(* Logix 5000 project; controller NSH_PLC2 vendor 1 type 14 code 167 rev 32.14; software revision 32.03; part 6 of 6 *)
(* tags used below, declared in another part *)
   AFI : BOOL;   // Always False
   AOI_PLC1_To_MCC3_10A : MotorToE300;
   AOI_PLC1_To_MCC3_10D : MotorToE300;
   AOI_PLC1_To_MCC3_10G : MotorToE300;
   AOI_PLC1_To_MCC3_10J : MotorToE300;
   AOI_PLC1_To_MCC3_11A : MotorToE300;
   AOI_PLC1_To_MCC3_11D : MotorToE300;
   AOI_PLC1_To_MCC3_11G : MotorToE300;
   AOI_PLC1_To_MCC3_11J : MotorToE300;
   AOI_PLC1_To_MCC3_12A : MotorToE300;
   AOI_PLC1_To_MCC3_12C : MotorToE300;
   AOI_PLC1_To_MCC3_12E : MotorToE300;
   AOI_PLC1_To_MCC3_12G : MotorToE300;
   AOI_PLC1_To_MCC3_12J : MotorToE300;
   AOI_PLC1_To_MCC3_12L : MotorToE300;
   AOI_PLC1_To_MCC3_13A : MotorToE300;
   AOI_PLC1_To_MCC3_13C : MotorToE300;
   AOI_PLC1_To_MCC3_13E : MotorToE300;
   AOI_PLC1_To_MCC3_13G : MotorToE300;
   AOI_PLC1_To_MCC3_13J : MotorToE300;
   AOI_PLC1_To_MCC3_13L : MotorToE300;
   AOI_PLC1_To_MCC3_14A : MotorToE300;
   AOI_PLC1_To_MCC3_14C : MotorToE300;
   AOI_PLC1_To_MCC3_14E : MotorToE300;
   AOI_PLC1_To_MCC3_14G : MotorToE300;
   AOI_PLC1_To_MCC3_14J : MotorToE300;
   AOI_PLC1_To_MCC3_14L : MotorToE300;
   AOI_PLC1_To_MCC3_15A : MotorToE300;
   AOI_PLC1_To_MCC3_15C : MotorToE300;
   AOI_PLC1_To_MCC3_15E : MotorToE300;
   AOI_PLC1_To_MCC3_15G : MotorToE300;
   AOI_PLC1_To_MCC3_15J : MotorToE300;
   AOI_PLC1_To_MCC3_16A : MotorToE300;
   AOI_PLC1_To_MCC3_16C : MotorToE300;
   AOI_PLC1_To_MCC3_16E : MotorToE300;
   AOI_PLC1_To_MCC3_16G : MotorToE300;
   AOI_PLC1_To_MCC3_16J : MotorToE300;
   AOI_PLC1_To_MCC3_16L : MotorToE300;
   AOI_PLC1_To_MCC3_17A : MotorToE300;
   AOI_PLC1_To_MCC3_17C : MotorToE300;
   AOI_PLC1_To_MCC3_17E : MotorToE300;
   AOI_PLC1_To_MCC3_17G : MotorToE300;
   AOI_PLC1_To_MCC3_17J : MotorToE300;
   AOI_PLC1_To_MCC3_17L : MotorToE300;
   AOI_PLC1_To_MCC3_18A : MotorToE300;
   AOI_PLC1_To_MCC3_18C : MotorToE300;
   AOI_PLC1_To_MCC3_18E : MotorToE300;
   AOI_PLC1_To_MCC3_18G : MotorToE300;
   AOI_PLC1_To_MCC3_18J : MotorToE300;
   AOI_PLC1_To_MCC3_18L : MotorToE300;
   AOI_PLC1_To_MCC3_19A : MotorToE300;
   AOI_PLC1_To_MCC3_19C : MotorToE300;
   AOI_PLC1_To_MCC3_19E : MotorToE300;
   AOI_PLC1_To_MCC3_19G : MotorToE300;
   AOI_PLC1_To_MCC3_19J : MotorToE300;
   AOI_PLC1_To_MCC3_20A : MotorToE300;
   AOI_PLC1_To_MCC3_20C : MotorToE300;
   AOI_PLC1_To_MCC3_20E : MotorToE300;
   AOI_PLC1_To_MCC3_20G : MotorToE300;
   AOI_PLC1_To_MCC3_20J : MotorToE300;
   AOI_PLC1_To_MCC3_21A : MotorToE300;
   AOI_PLC1_To_MCC3_21C : MotorToE300;
   AOI_PLC1_To_MCC3_21E : MotorToE300;
   AOI_PLC1_To_MCC3_21G : MotorToE300;
   AOI_PLC1_To_MCC3_21J : MotorToE300;
   AOI_PLC1_To_MCC3_21L : MotorToE300;
   AOI_PLC1_To_MCC3_22C : MotorToE300;
   AOI_PLC1_To_MCC3_22E : MotorToE300;
   AOI_PLC1_To_MCC3_7A : MotorToE300;
   AOI_PLC1_To_MCC3_7C : MotorToE300;
   AOI_PLC1_To_MCC3_7E : MotorToE300;
   AOI_PLC1_To_MCC3_7G : MotorToPF525;
   AOI_PLC1_To_MCC3_7K : MotorToPF525;
   AOI_PLC1_To_MCC3_8A : MotorToE300;
   AOI_PLC1_To_MCC3_8D : MotorToPF525;
   AOI_PLC1_To_MCC3_8H : MotorToE300;
   AOI_PLC1_To_MCC3_8K : MotorToPF525;
   AOI_PLC1_To_MCC3_9A : MotorToE300;
   AOI_PLC1_To_MCC3_9C : MotorToE300;
   AOI_PLC1_To_MCC3_9E : MotorToE300;
   AOI_PLC1_To_MCC3_9G : MotorToE300;
   AOI_PLC1_To_MCC3_9J : MotorToE300;
   AOI_PLC1_To_MCC3_9L : MotorToE300;
   AOI_PLC1_To_MCC4_1E : MotorToPF525;
   AOI_PLC1_To_MCC4_2A : MotorToE300;
   AOI_PLC1_To_MCC4_2C : MotorToE300;
   AOI_PLC1_To_MCC4_2E : MotorToE300;
   AOI_PLC1_To_MCC4_2G : MotorToPF525;
   AOI_PLC1_To_MCC4_2K : MotorToPF525;
   AOI_PLC1_To_MCC4_3A : MotorToE300;
   AOI_PLC1_To_MCC4_3C : MotorToE300;
   AOI_PLC1_To_MCC4_3E : MotorToE300;
   AOI_PLC1_To_MCC4_3G : MotorToE300;
   AOI_PLC1_To_MCC4_3J : MotorToE300;
   AOI_PLC1_To_MCC4_3L : MotorToE300;
   AOI_PLC1_To_MCC4_4A : MotorToE300;
   AOI_PLC1_To_MCC4_4C : MotorToE300;
   AOI_PLC1_To_MCC4_4E : MotorToE300;
   AOI_PLC1_To_MCC4_4G : MotorToE300;
   AOI_PLC1_To_MCC4_4J : MotorToE300;
   AOI_PLC1_To_MCC4_4L : MotorToE300;
   AOI_PLC1_To_MCC4_5A : MotorToE300;
   AOI_PLC1_To_MCC4_5C : MotorToE300;
   MotorsControlTag : MotorsControlUDT;   // Only Instance of UDT
   OKToRunMotors : BOOL;   // Messages from PLC1 Ok, OK to run
(* MainProgram, continued *)

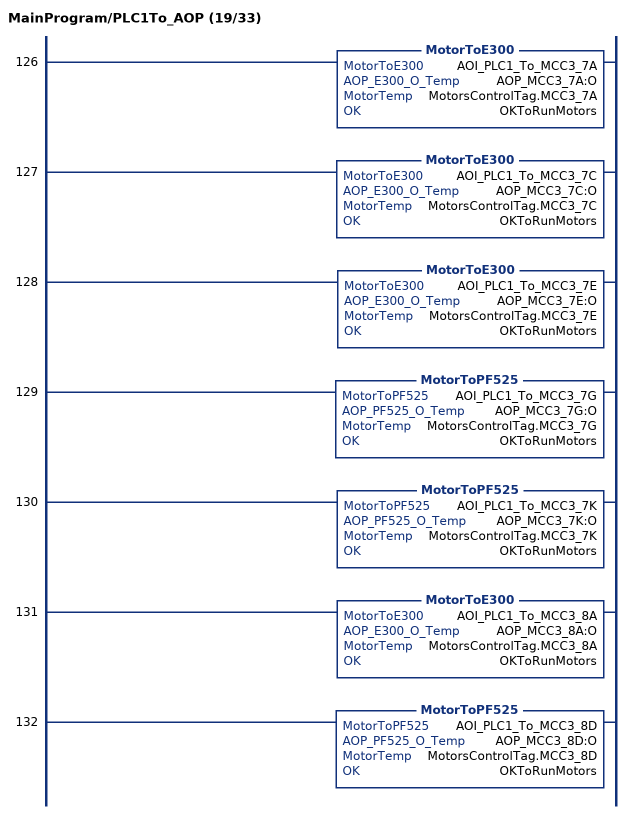
   [picture p103: MainProgram/PLC1To_AOP rungs 126-132]
   126: MotorToE300(AOI_PLC1_To_MCC3_7A,AOP_MCC3_7A:O,MotorsControlTag.MCC3_7A,OKToRunMotors);
   127: MotorToE300(AOI_PLC1_To_MCC3_7C,AOP_MCC3_7C:O,MotorsControlTag.MCC3_7C,OKToRunMotors);
   128: MotorToE300(AOI_PLC1_To_MCC3_7E,AOP_MCC3_7E:O,MotorsControlTag.MCC3_7E,OKToRunMotors);
   129: MotorToPF525(AOI_PLC1_To_MCC3_7G,AOP_MCC3_7G:O,MotorsControlTag.MCC3_7G,OKToRunMotors);
   130: MotorToPF525(AOI_PLC1_To_MCC3_7K,AOP_MCC3_7K:O,MotorsControlTag.MCC3_7K,OKToRunMotors);
   131: MotorToE300(AOI_PLC1_To_MCC3_8A,AOP_MCC3_8A:O,MotorsControlTag.MCC3_8A,OKToRunMotors);
   132: MotorToPF525(AOI_PLC1_To_MCC3_8D,AOP_MCC3_8D:O,MotorsControlTag.MCC3_8D,OKToRunMotors);
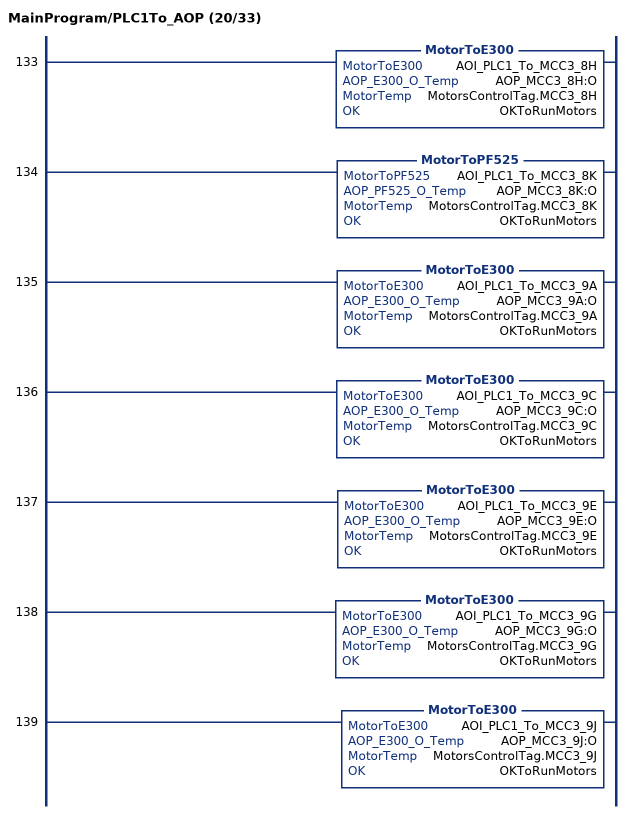
   133: MotorToE300(AOI_PLC1_To_MCC3_8H,AOP_MCC3_8H:O,MotorsControlTag.MCC3_8H,OKToRunMotors);
   134: MotorToPF525(AOI_PLC1_To_MCC3_8K,AOP_MCC3_8K:O,MotorsControlTag.MCC3_8K,OKToRunMotors);
   135: MotorToE300(AOI_PLC1_To_MCC3_9A,AOP_MCC3_9A:O,MotorsControlTag.MCC3_9A,OKToRunMotors);
   136: MotorToE300(AOI_PLC1_To_MCC3_9C,AOP_MCC3_9C:O,MotorsControlTag.MCC3_9C,OKToRunMotors);
   137: MotorToE300(AOI_PLC1_To_MCC3_9E,AOP_MCC3_9E:O,MotorsControlTag.MCC3_9E,OKToRunMotors);
   138: MotorToE300(AOI_PLC1_To_MCC3_9G,AOP_MCC3_9G:O,MotorsControlTag.MCC3_9G,OKToRunMotors);
   139: MotorToE300(AOI_PLC1_To_MCC3_9J,AOP_MCC3_9J:O,MotorsControlTag.MCC3_9J,OKToRunMotors);
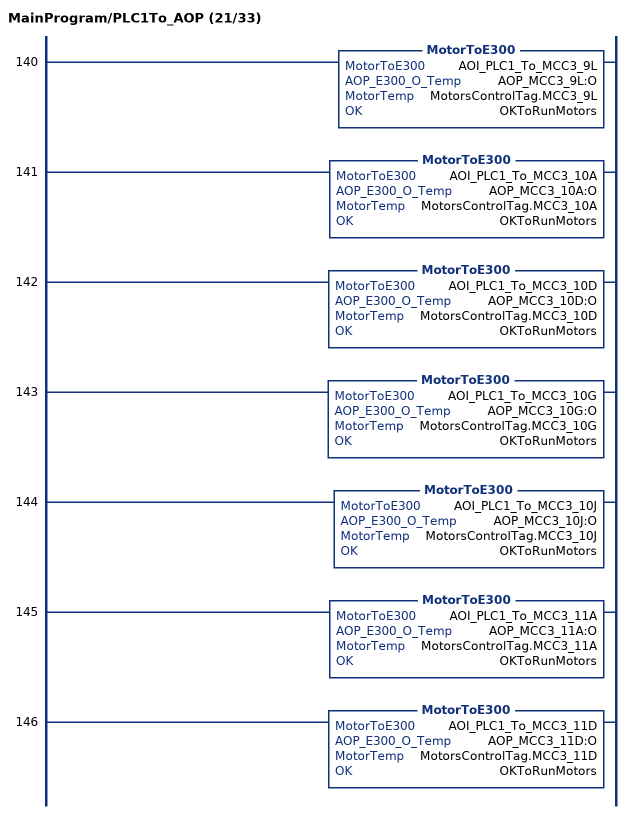
   140: MotorToE300(AOI_PLC1_To_MCC3_9L,AOP_MCC3_9L:O,MotorsControlTag.MCC3_9L,OKToRunMotors);
   141: MotorToE300(AOI_PLC1_To_MCC3_10A,AOP_MCC3_10A:O,MotorsControlTag.MCC3_10A,OKToRunMotors);
   142: MotorToE300(AOI_PLC1_To_MCC3_10D,AOP_MCC3_10D:O,MotorsControlTag.MCC3_10D,OKToRunMotors);
   143: MotorToE300(AOI_PLC1_To_MCC3_10G,AOP_MCC3_10G:O,MotorsControlTag.MCC3_10G,OKToRunMotors);
   144: MotorToE300(AOI_PLC1_To_MCC3_10J,AOP_MCC3_10J:O,MotorsControlTag.MCC3_10J,OKToRunMotors);
   145: MotorToE300(AOI_PLC1_To_MCC3_11A,AOP_MCC3_11A:O,MotorsControlTag.MCC3_11A,OKToRunMotors);
   146: MotorToE300(AOI_PLC1_To_MCC3_11D,AOP_MCC3_11D:O,MotorsControlTag.MCC3_11D,OKToRunMotors);
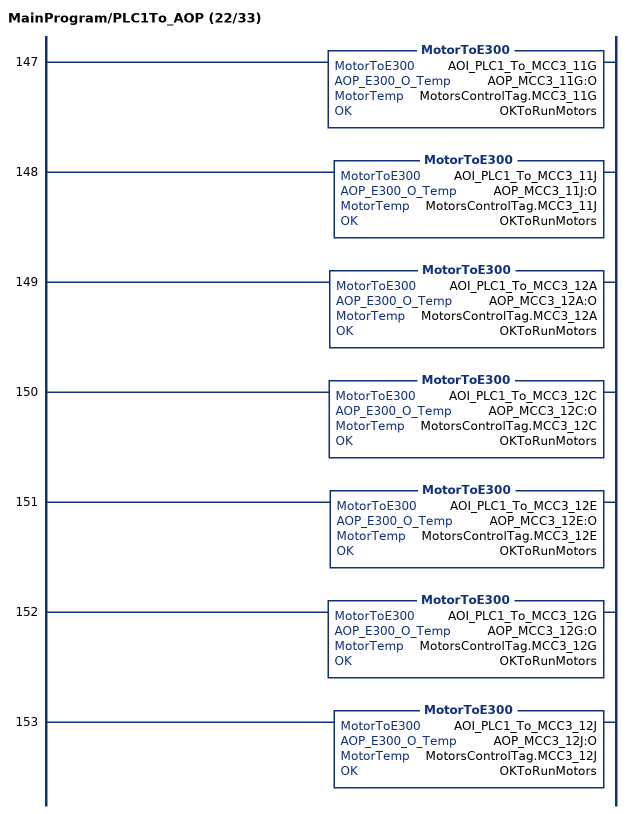
   147: MotorToE300(AOI_PLC1_To_MCC3_11G,AOP_MCC3_11G:O,MotorsControlTag.MCC3_11G,OKToRunMotors);
   148: MotorToE300(AOI_PLC1_To_MCC3_11J,AOP_MCC3_11J:O,MotorsControlTag.MCC3_11J,OKToRunMotors);
   149: MotorToE300(AOI_PLC1_To_MCC3_12A,AOP_MCC3_12A:O,MotorsControlTag.MCC3_12A,OKToRunMotors);
   150: MotorToE300(AOI_PLC1_To_MCC3_12C,AOP_MCC3_12C:O,MotorsControlTag.MCC3_12C,OKToRunMotors);
   151: MotorToE300(AOI_PLC1_To_MCC3_12E,AOP_MCC3_12E:O,MotorsControlTag.MCC3_12E,OKToRunMotors);
   152: MotorToE300(AOI_PLC1_To_MCC3_12G,AOP_MCC3_12G:O,MotorsControlTag.MCC3_12G,OKToRunMotors);
   153: MotorToE300(AOI_PLC1_To_MCC3_12J,AOP_MCC3_12J:O,MotorsControlTag.MCC3_12J,OKToRunMotors);
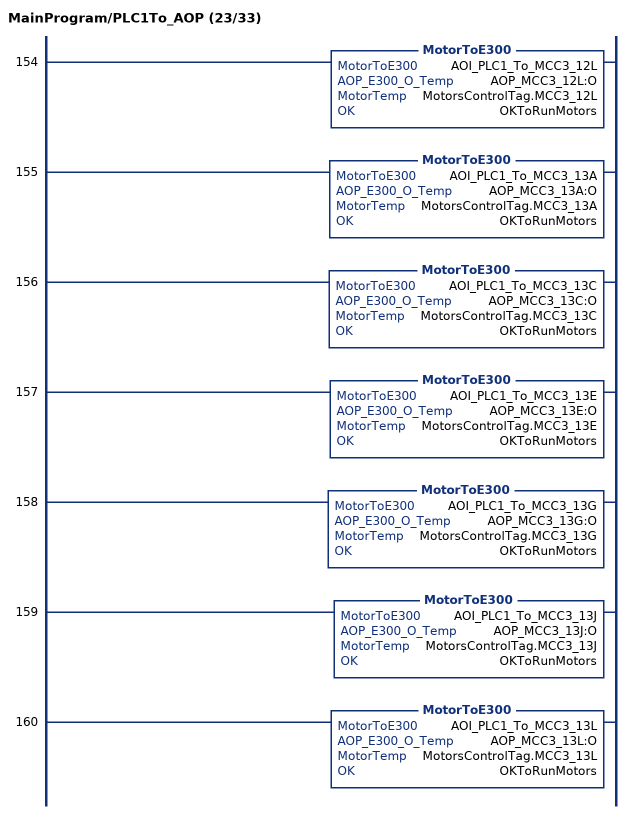
   154: MotorToE300(AOI_PLC1_To_MCC3_12L,AOP_MCC3_12L:O,MotorsControlTag.MCC3_12L,OKToRunMotors);
   155: MotorToE300(AOI_PLC1_To_MCC3_13A,AOP_MCC3_13A:O,MotorsControlTag.MCC3_13A,OKToRunMotors);
   156: MotorToE300(AOI_PLC1_To_MCC3_13C,AOP_MCC3_13C:O,MotorsControlTag.MCC3_13C,OKToRunMotors);
   157: MotorToE300(AOI_PLC1_To_MCC3_13E,AOP_MCC3_13E:O,MotorsControlTag.MCC3_13E,OKToRunMotors);
   158: MotorToE300(AOI_PLC1_To_MCC3_13G,AOP_MCC3_13G:O,MotorsControlTag.MCC3_13G,OKToRunMotors);
   159: MotorToE300(AOI_PLC1_To_MCC3_13J,AOP_MCC3_13J:O,MotorsControlTag.MCC3_13J,OKToRunMotors);
   160: MotorToE300(AOI_PLC1_To_MCC3_13L,AOP_MCC3_13L:O,MotorsControlTag.MCC3_13L,OKToRunMotors);
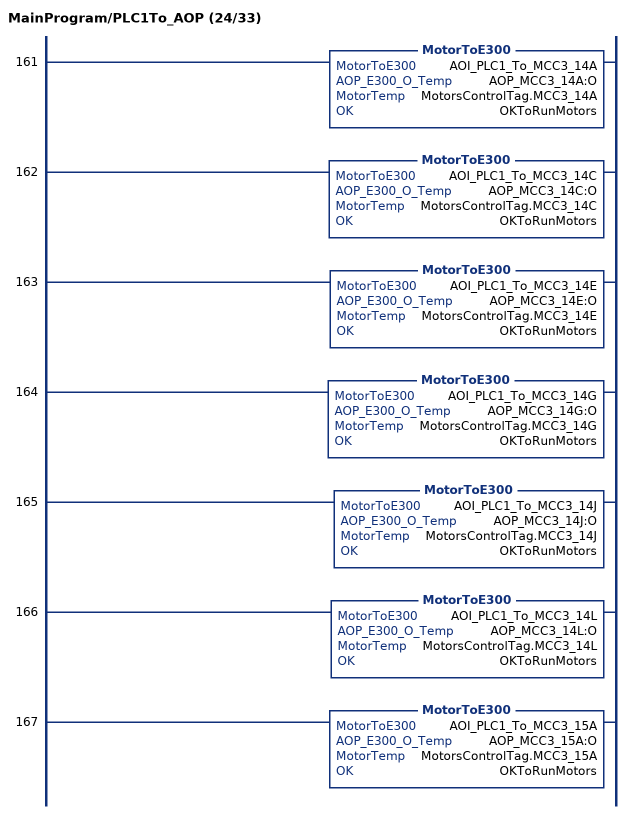
   161: MotorToE300(AOI_PLC1_To_MCC3_14A,AOP_MCC3_14A:O,MotorsControlTag.MCC3_14A,OKToRunMotors);
   162: MotorToE300(AOI_PLC1_To_MCC3_14C,AOP_MCC3_14C:O,MotorsControlTag.MCC3_14C,OKToRunMotors);
   163: MotorToE300(AOI_PLC1_To_MCC3_14E,AOP_MCC3_14E:O,MotorsControlTag.MCC3_14E,OKToRunMotors);
   164: MotorToE300(AOI_PLC1_To_MCC3_14G,AOP_MCC3_14G:O,MotorsControlTag.MCC3_14G,OKToRunMotors);
   165: MotorToE300(AOI_PLC1_To_MCC3_14J,AOP_MCC3_14J:O,MotorsControlTag.MCC3_14J,OKToRunMotors);
   166: MotorToE300(AOI_PLC1_To_MCC3_14L,AOP_MCC3_14L:O,MotorsControlTag.MCC3_14L,OKToRunMotors);
   167: MotorToE300(AOI_PLC1_To_MCC3_15A,AOP_MCC3_15A:O,MotorsControlTag.MCC3_15A,OKToRunMotors);
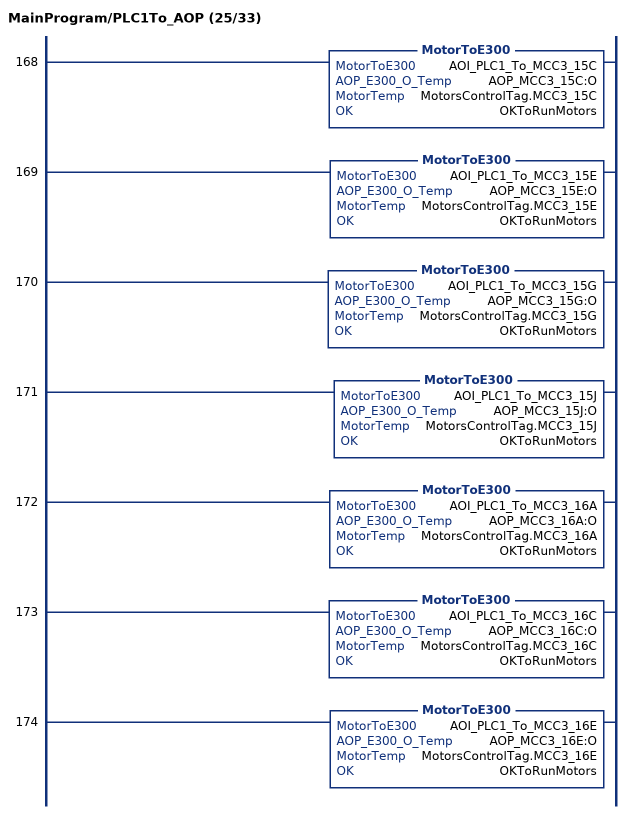
   168: MotorToE300(AOI_PLC1_To_MCC3_15C,AOP_MCC3_15C:O,MotorsControlTag.MCC3_15C,OKToRunMotors);
   169: MotorToE300(AOI_PLC1_To_MCC3_15E,AOP_MCC3_15E:O,MotorsControlTag.MCC3_15E,OKToRunMotors);
   170: MotorToE300(AOI_PLC1_To_MCC3_15G,AOP_MCC3_15G:O,MotorsControlTag.MCC3_15G,OKToRunMotors);
   171: MotorToE300(AOI_PLC1_To_MCC3_15J,AOP_MCC3_15J:O,MotorsControlTag.MCC3_15J,OKToRunMotors);
   172: MotorToE300(AOI_PLC1_To_MCC3_16A,AOP_MCC3_16A:O,MotorsControlTag.MCC3_16A,OKToRunMotors);
   173: MotorToE300(AOI_PLC1_To_MCC3_16C,AOP_MCC3_16C:O,MotorsControlTag.MCC3_16C,OKToRunMotors);
   174: MotorToE300(AOI_PLC1_To_MCC3_16E,AOP_MCC3_16E:O,MotorsControlTag.MCC3_16E,OKToRunMotors);
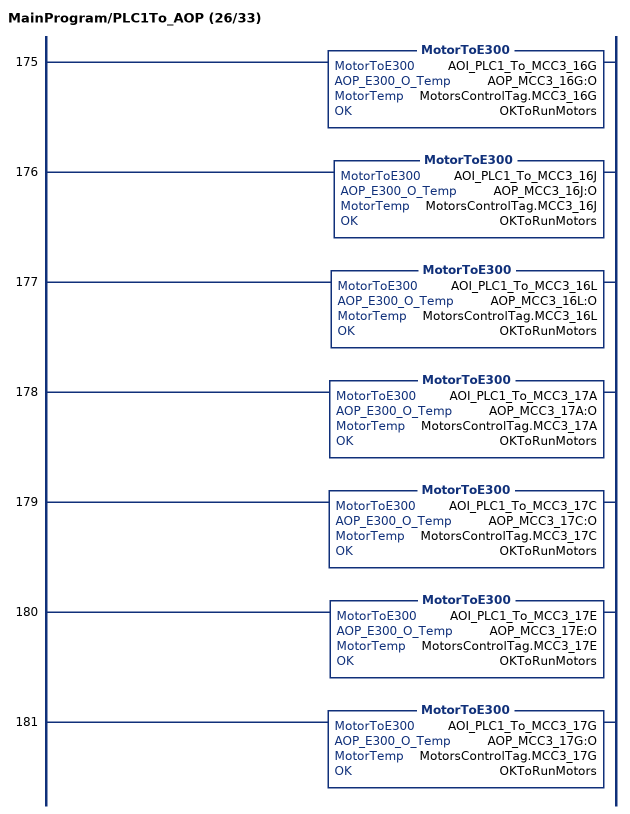
   175: MotorToE300(AOI_PLC1_To_MCC3_16G,AOP_MCC3_16G:O,MotorsControlTag.MCC3_16G,OKToRunMotors);
   176: MotorToE300(AOI_PLC1_To_MCC3_16J,AOP_MCC3_16J:O,MotorsControlTag.MCC3_16J,OKToRunMotors);
   177: MotorToE300(AOI_PLC1_To_MCC3_16L,AOP_MCC3_16L:O,MotorsControlTag.MCC3_16L,OKToRunMotors);
   178: MotorToE300(AOI_PLC1_To_MCC3_17A,AOP_MCC3_17A:O,MotorsControlTag.MCC3_17A,OKToRunMotors);
   179: MotorToE300(AOI_PLC1_To_MCC3_17C,AOP_MCC3_17C:O,MotorsControlTag.MCC3_17C,OKToRunMotors);
   180: MotorToE300(AOI_PLC1_To_MCC3_17E,AOP_MCC3_17E:O,MotorsControlTag.MCC3_17E,OKToRunMotors);
   181: MotorToE300(AOI_PLC1_To_MCC3_17G,AOP_MCC3_17G:O,MotorsControlTag.MCC3_17G,OKToRunMotors);
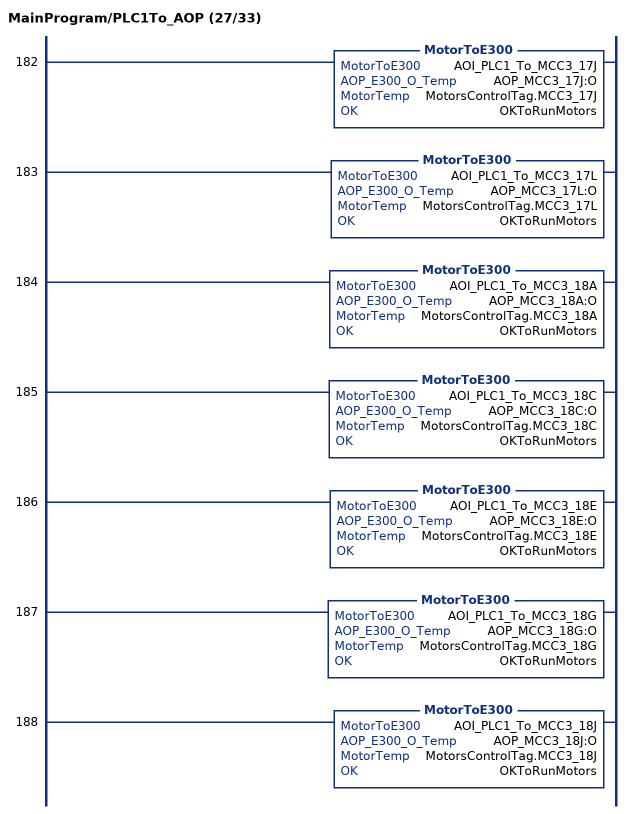
   182: MotorToE300(AOI_PLC1_To_MCC3_17J,AOP_MCC3_17J:O,MotorsControlTag.MCC3_17J,OKToRunMotors);
   183: MotorToE300(AOI_PLC1_To_MCC3_17L,AOP_MCC3_17L:O,MotorsControlTag.MCC3_17L,OKToRunMotors);
   184: MotorToE300(AOI_PLC1_To_MCC3_18A,AOP_MCC3_18A:O,MotorsControlTag.MCC3_18A,OKToRunMotors);
   185: MotorToE300(AOI_PLC1_To_MCC3_18C,AOP_MCC3_18C:O,MotorsControlTag.MCC3_18C,OKToRunMotors);
   186: MotorToE300(AOI_PLC1_To_MCC3_18E,AOP_MCC3_18E:O,MotorsControlTag.MCC3_18E,OKToRunMotors);
   187: MotorToE300(AOI_PLC1_To_MCC3_18G,AOP_MCC3_18G:O,MotorsControlTag.MCC3_18G,OKToRunMotors);
   188: MotorToE300(AOI_PLC1_To_MCC3_18J,AOP_MCC3_18J:O,MotorsControlTag.MCC3_18J,OKToRunMotors);
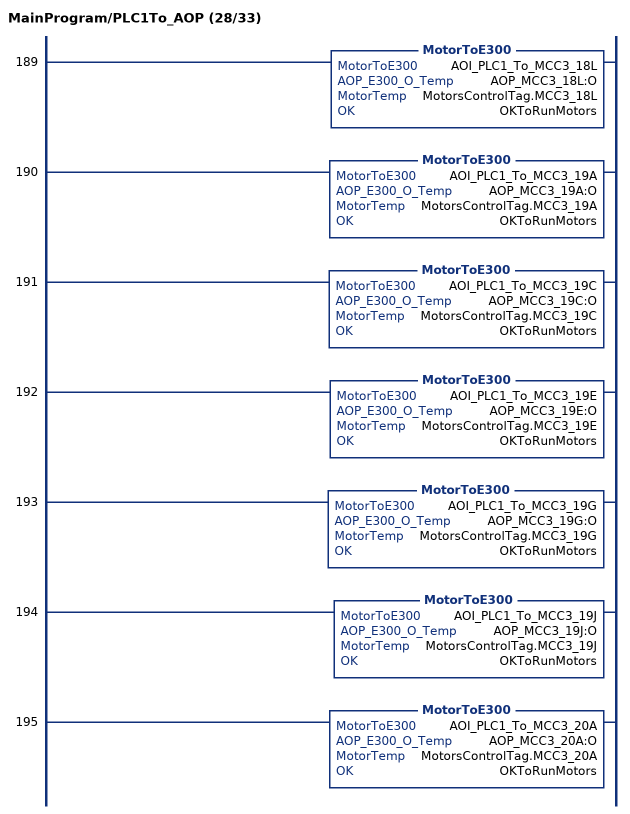
   189: MotorToE300(AOI_PLC1_To_MCC3_18L,AOP_MCC3_18L:O,MotorsControlTag.MCC3_18L,OKToRunMotors);
   190: MotorToE300(AOI_PLC1_To_MCC3_19A,AOP_MCC3_19A:O,MotorsControlTag.MCC3_19A,OKToRunMotors);
   191: MotorToE300(AOI_PLC1_To_MCC3_19C,AOP_MCC3_19C:O,MotorsControlTag.MCC3_19C,OKToRunMotors);
   192: MotorToE300(AOI_PLC1_To_MCC3_19E,AOP_MCC3_19E:O,MotorsControlTag.MCC3_19E,OKToRunMotors);
   193: MotorToE300(AOI_PLC1_To_MCC3_19G,AOP_MCC3_19G:O,MotorsControlTag.MCC3_19G,OKToRunMotors);
   194: MotorToE300(AOI_PLC1_To_MCC3_19J,AOP_MCC3_19J:O,MotorsControlTag.MCC3_19J,OKToRunMotors);
   195: MotorToE300(AOI_PLC1_To_MCC3_20A,AOP_MCC3_20A:O,MotorsControlTag.MCC3_20A,OKToRunMotors);
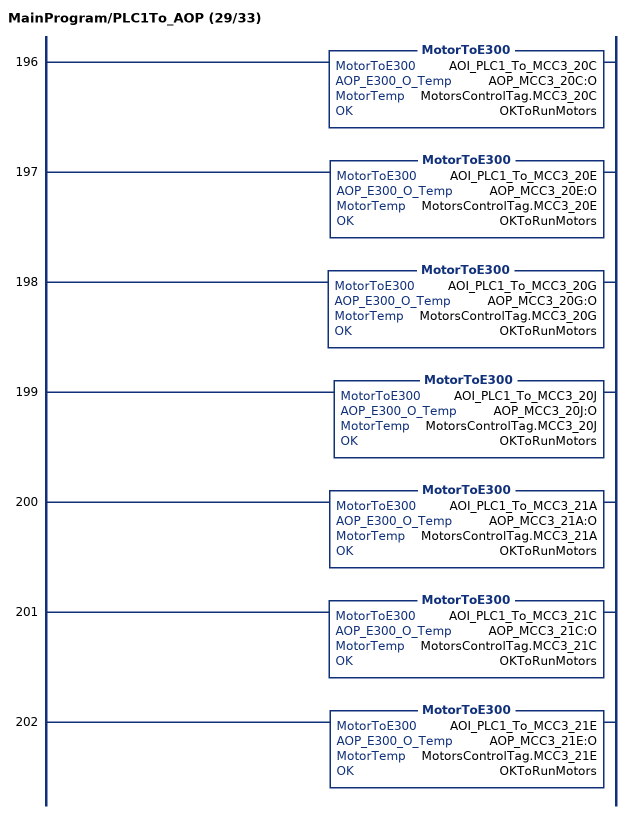
   196: MotorToE300(AOI_PLC1_To_MCC3_20C,AOP_MCC3_20C:O,MotorsControlTag.MCC3_20C,OKToRunMotors);
   197: MotorToE300(AOI_PLC1_To_MCC3_20E,AOP_MCC3_20E:O,MotorsControlTag.MCC3_20E,OKToRunMotors);
   198: MotorToE300(AOI_PLC1_To_MCC3_20G,AOP_MCC3_20G:O,MotorsControlTag.MCC3_20G,OKToRunMotors);
   199: MotorToE300(AOI_PLC1_To_MCC3_20J,AOP_MCC3_20J:O,MotorsControlTag.MCC3_20J,OKToRunMotors);
   200: MotorToE300(AOI_PLC1_To_MCC3_21A,AOP_MCC3_21A:O,MotorsControlTag.MCC3_21A,OKToRunMotors);
   201: MotorToE300(AOI_PLC1_To_MCC3_21C,AOP_MCC3_21C:O,MotorsControlTag.MCC3_21C,OKToRunMotors);
   202: MotorToE300(AOI_PLC1_To_MCC3_21E,AOP_MCC3_21E:O,MotorsControlTag.MCC3_21E,OKToRunMotors);
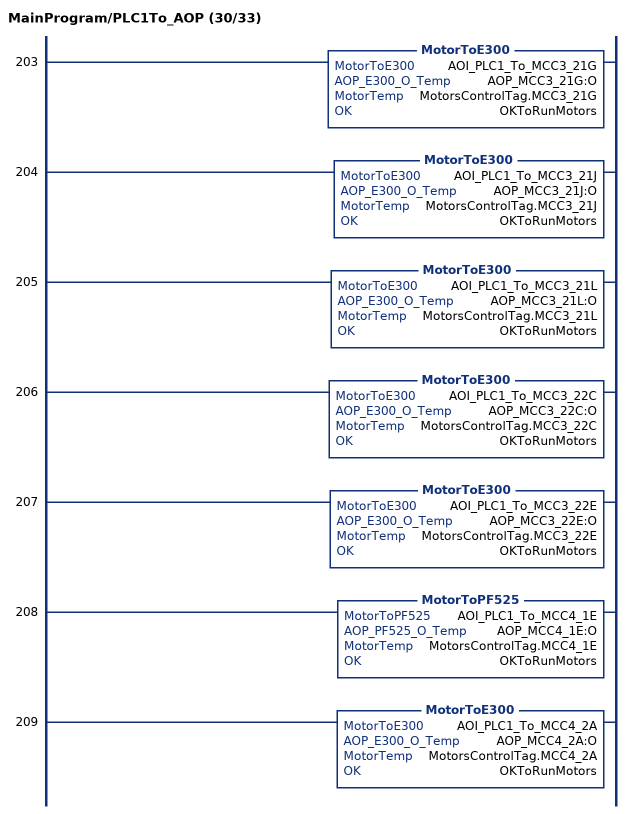
   203: MotorToE300(AOI_PLC1_To_MCC3_21G,AOP_MCC3_21G:O,MotorsControlTag.MCC3_21G,OKToRunMotors);
   204: MotorToE300(AOI_PLC1_To_MCC3_21J,AOP_MCC3_21J:O,MotorsControlTag.MCC3_21J,OKToRunMotors);
   205: MotorToE300(AOI_PLC1_To_MCC3_21L,AOP_MCC3_21L:O,MotorsControlTag.MCC3_21L,OKToRunMotors);
   206: MotorToE300(AOI_PLC1_To_MCC3_22C,AOP_MCC3_22C:O,MotorsControlTag.MCC3_22C,OKToRunMotors);
   207: MotorToE300(AOI_PLC1_To_MCC3_22E,AOP_MCC3_22E:O,MotorsControlTag.MCC3_22E,OKToRunMotors);
   208: MotorToPF525(AOI_PLC1_To_MCC4_1E,AOP_MCC4_1E:O,MotorsControlTag.MCC4_1E,OKToRunMotors);
   209: MotorToE300(AOI_PLC1_To_MCC4_2A,AOP_MCC4_2A:O,MotorsControlTag.MCC4_2A,OKToRunMotors);
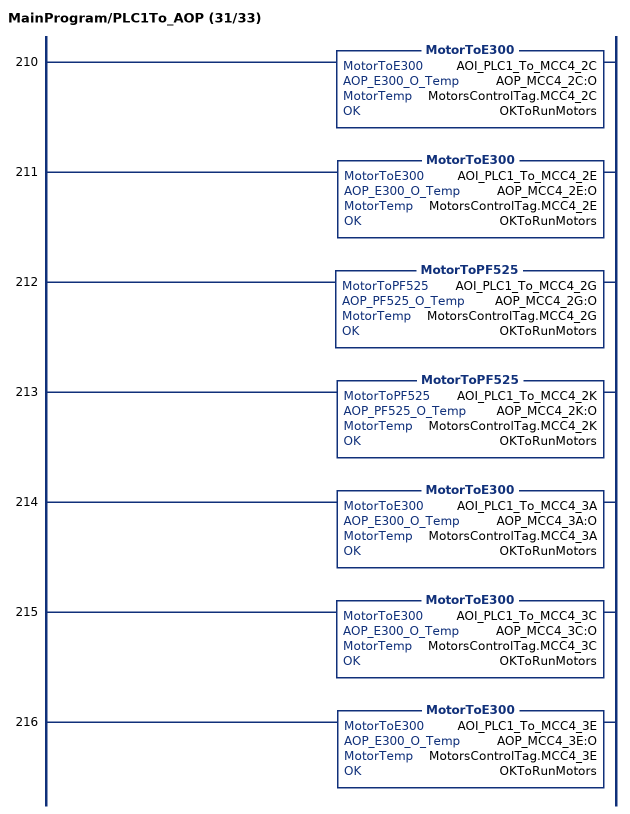
   210: MotorToE300(AOI_PLC1_To_MCC4_2C,AOP_MCC4_2C:O,MotorsControlTag.MCC4_2C,OKToRunMotors);
   211: MotorToE300(AOI_PLC1_To_MCC4_2E,AOP_MCC4_2E:O,MotorsControlTag.MCC4_2E,OKToRunMotors);
   212: MotorToPF525(AOI_PLC1_To_MCC4_2G,AOP_MCC4_2G:O,MotorsControlTag.MCC4_2G,OKToRunMotors);
   213: MotorToPF525(AOI_PLC1_To_MCC4_2K,AOP_MCC4_2K:O,MotorsControlTag.MCC4_2K,OKToRunMotors);
   214: MotorToE300(AOI_PLC1_To_MCC4_3A,AOP_MCC4_3A:O,MotorsControlTag.MCC4_3A,OKToRunMotors);
   215: MotorToE300(AOI_PLC1_To_MCC4_3C,AOP_MCC4_3C:O,MotorsControlTag.MCC4_3C,OKToRunMotors);
   216: MotorToE300(AOI_PLC1_To_MCC4_3E,AOP_MCC4_3E:O,MotorsControlTag.MCC4_3E,OKToRunMotors);
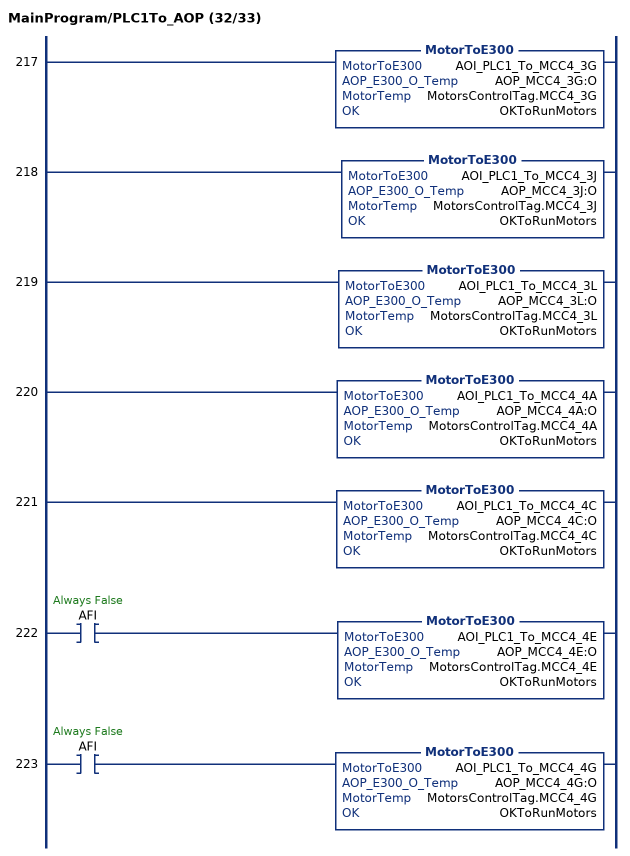
   217: MotorToE300(AOI_PLC1_To_MCC4_3G,AOP_MCC4_3G:O,MotorsControlTag.MCC4_3G,OKToRunMotors);
   218: MotorToE300(AOI_PLC1_To_MCC4_3J,AOP_MCC4_3J:O,MotorsControlTag.MCC4_3J,OKToRunMotors);
   219: MotorToE300(AOI_PLC1_To_MCC4_3L,AOP_MCC4_3L:O,MotorsControlTag.MCC4_3L,OKToRunMotors);
   220: MotorToE300(AOI_PLC1_To_MCC4_4A,AOP_MCC4_4A:O,MotorsControlTag.MCC4_4A,OKToRunMotors);
   221: MotorToE300(AOI_PLC1_To_MCC4_4C,AOP_MCC4_4C:O,MotorsControlTag.MCC4_4C,OKToRunMotors);
   222: XIC(AFI)MotorToE300(AOI_PLC1_To_MCC4_4E,AOP_MCC4_4E:O,MotorsControlTag.MCC4_4E,OKToRunMotors);
   223: XIC(AFI)MotorToE300(AOI_PLC1_To_MCC4_4G,AOP_MCC4_4G:O,MotorsControlTag.MCC4_4G,OKToRunMotors);
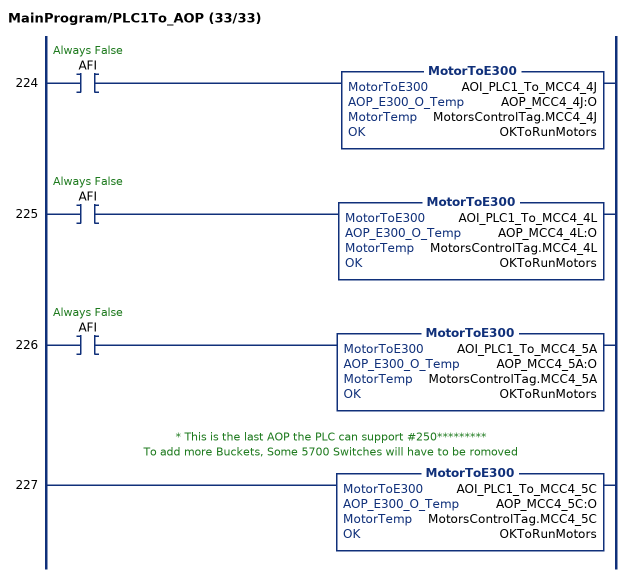
   224: XIC(AFI)MotorToE300(AOI_PLC1_To_MCC4_4J,AOP_MCC4_4J:O,MotorsControlTag.MCC4_4J,OKToRunMotors);
   225: XIC(AFI)MotorToE300(AOI_PLC1_To_MCC4_4L,AOP_MCC4_4L:O,MotorsControlTag.MCC4_4L,OKToRunMotors);
   226: XIC(AFI)MotorToE300(AOI_PLC1_To_MCC4_5A,AOP_MCC4_5A:O,MotorsControlTag.MCC4_5A,OKToRunMotors);
   // * This is the last AOP the PLC can support #250*********
   // To add more Buckets, Some 5700 Switches will have to be romoved
   227: MotorToE300(AOI_PLC1_To_MCC4_5C,AOP_MCC4_5C:O,MotorsControlTag.MCC4_5C,OKToRunMotors);
END_ROUTINE
END_PROGRAM
